// TwinCAT 3 PLC project TimerExample
// ProgramVersion: 3.1.4023.0
// libraries:
//   Tc2_Standard, * (Beckhoff Automation GmbH)
//   Tc2_System, * (Beckhoff Automation GmbH)
//   Tc3_Module, * (Beckhoff Automation GmbH)
//   VisuSymbols,3.5.10.0,System
// project tree:
//   / GlobalTextList.TcGTLO, PlcTask.TcTTO, Visualisierungsmanager.TcVMO (not stored)
//   GVLs/ I0.TcGVL, IO.TcDUT
//   POUs/ fb_EdgeDetector.TcPOU, MAIN.TcPOU
//   VISUs/ Visualization.TcVIS
// (motion and I/O tree: see PLC project aufgabensammlung2)
// real-time tasks:
//   TASK PlcTask: cycle T#10ms, priority 20, ADS port 350
//   TASK PlcTask1: cycle T#10ms, priority 21, ADS port 351

CONFIGURATION TimerExample
    RESOURCE PLC ON TwinCAT3
        TASK PlcTask(INTERVAL := T#10ms, PRIORITY := 21);
        PROGRAM MAIN WITH PlcTask : MAIN;
    END_RESOURCE
END_CONFIGURATION

// ---- GVLs/IO.TcDUT
TYPE  IO :
STRUCT
	bLampeGruen		:	BOOL;
	bLampeGelb		:	BOOL;
	bLampeRot		:	BOOL;
	
	bSchalterBlau	:	BOOL;
	bSchalterGelb	:	BOOL;
END_STRUCT
END_TYPE

// ---- GVLs/I0.TcGVL
{attribute 'qualified_only'}
VAR_GLOBAL
	bLampeGruen		:	BOOL;
	bLampeGelb		:	BOOL;
	bLampeRot		:	BOOL;
	
	bSchalterBlau	:	BOOL;
	bSchalterGelb	:	BOOL;
END_VAR

// ---- POUs/MAIN.TcPOU
PROGRAM MAIN
VAR	

	FB_EdgeDetector1	: fb_EdgeDetector;
	FB_EdgeDetector2	: fb_EdgeDetector;
	bTaster 			: BOOL;
	timeDelay			: TIME := T#200MS;
	bRising				: BOOL;
	bFalling			: BOOL;
	bOldState			: BOOL;
END_VAR

FB_EdgeDetector1(bSignal := I0.bSchalterBlau, timeON := timeDelay, bRisingEdge =>bRising, bFallingEdge =>bFalling);
IF bRising  THEN
	IF bOldState THEN
		bOldState := FALSE;
		I0.bLampeGelb := TRUE;
	ELSE
		bOldState := TRUE;
		I0.bLampeGelb := FALSE;
	END_IF
END_IF

END_PROGRAM

// ---- POUs/fb_EdgeDetector.TcPOU
FUNCTION_BLOCK fb_EdgeDetector
VAR_INPUT
	bSignal			:	BOOL;
	timeON			:	TIME := T#200MS;
	bDoupleTap		:	BOOL;
	timeDoubleTap	: 	TIME := T#200MS;
END_VAR
VAR_OUTPUT
	bRisingEdge		:	BOOL;
	bFallingEdge	: 	BOOL;
END_VAR
VAR
	timer			:	TON;
	bOnMeasure		:	BOOL;
	bOldState		: 	BOOL;
END_VAR

// set default state
timer.IN 	:= TRUE;
bRisingEdge	:= FALSE;
bFallingEdge:= FALSE;
timer.PT	:= timeON;
IF bSignal THEN
	IF NOT bSignal =  bOldState THEN
		// State wechsel
		timer.IN := FALSE;
		bOnMeasure := TRUE;
	END_IF
	IF timer.Q AND bOnMeasure THEN
		bOnMeasure := FALSE;
		bRisingEdge := TRUE;
	END_IF
ELSE
	IF NOT bSignal =  bOldState THEN
		// State wechsle
		timer.IN := FALSE;
		bOnMeasure := TRUE;
	END_IF
	IF timer.Q AND bOnMeasure THEN
		bOnMeasure := FALSE;
		bFallingEdge := TRUE;
	END_IF
END_IF

timer();

END_FUNCTION_BLOCK

// ---- VISUs/Visualization.TcVIS
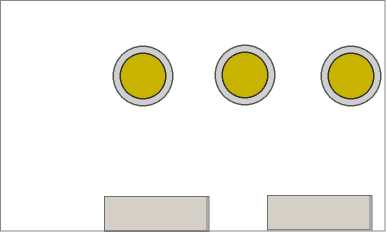
VISUALIZATION Visualization  // 386x232
    Lamp1 (108,41 70x70), variable: I0.bLampeGruen, style: Lamp-Lamp1-Yellow
    Lamp1 (210,40 70x70), variable: I0.bLampeGelb, style: Lamp-Lamp1-Yellow
    Lamp1 (316,41 70x70), variable: I0.bLampeRot, style: Lamp-Lamp1-Yellow
    Button (104,196 105x36)
        tap I0.bSchalterBlau
    Button (267,195 105x36)
        tap I0.bSchalterGelb
END_VISUALIZATION
